Fanuc KAREL source: remote_gripper_info.kl

PROGRAM remotegripperinfo

%COMMENT = ' Remote Gripper Info'
%NOLOCKGROUP
%NOPAUSE=ERROR+COMMAND+TPENABLE
%NOBUSYLAMP

CONST
	R_ABSDEPTH = 71
	R_RELDEPTH = 72
	R_WIDTH = 73
	R_ISBUSY = 74
	R_ISGRIP = 75
	R_ISSAFETY = 76
	R_ISCONNECT = 77

VAR
	temp_real: REAL
	temp_int: INTEGER

	abs_depth: REAL
	rel_depth: REAL
	width: REAL

	is_busy: INTEGER
	is_grip: INTEGER
	is_safety: INTEGER
	is_connect: INTEGER

	rf_ :FILE
	STATUS: INTEGER

BEGIN
	OPEN FILE rf_ ('RW', 'RD:RESPONSE.HTM')
	STATUS = IO_STATUS(rf_)
	IF (STATUS <> 0) THEN
		WRITE rf_ ( '{"result":"failed", "reason":',STATUS,'}')
		RETURN
	ENDIF

	-- abort current gripper instruction
	ABORT_TASK('gripper_info', TRUE, TRUE, STATUS)
	RUN_TASK( 'gripper_info', 1, FALSE, TRUE, 1 OR 2 OR 4, STATUS )
	DELAY(1) --yield

	IF (STATUS <> 0) THEN
		WRITE rf_ ( '{"result":"failed", "reason":',STATUS,'}')
		RETURN
	ENDIF

	GET_REG(R_ABSDEPTH, TRUE, temp_int, temp_real, STATUS)
	abs_depth = temp_real
	GET_REG(R_RELDEPTH, TRUE, temp_int, temp_real, STATUS)
	rel_depth = temp_real
	GET_REG(R_WIDTH, TRUE, temp_int, temp_real, STATUS)
	width= temp_real

	GET_REG(R_ISBUSY, FALSE, temp_int, temp_real, STATUS)
	is_busy = temp_int
	GET_REG(R_ISGRIP, FALSE, temp_int, temp_real, STATUS)
	is_grip = temp_int
	GET_REG(R_ISSAFETY, FALSE, temp_int, temp_real, STATUS)
	is_safety = temp_int
	GET_REG(R_ISCONNECT, FALSE, temp_int, temp_real, STATUS)
	is_connect = temp_int

	WRITE rf_ (  '{"result":"success"',
			', "abs_depth":',abs_depth ,
			', "rel_depth":',rel_depth ,
			', "width":', width,
			', "is_busy":',is_busy ,
			', "is_grip":',is_grip ,
			', "is_safety":',is_safety ,
			', "is_connect":',is_connect ,
			'}', CR)

	CLOSE FILE rf_
END remotegripperinfo
